FUNCTION_BLOCK FB_StartPos
VAR_INPUT
	bEnable 		: BOOL;
	fCurrentPos 	: LREAL;
END_VAR
VAR_OUTPUT
	fStartPos 		: LREAL;
END_VAR
VAR
END_VAR

IF bEnable THEN
	fStartPos := fStartPos;
	
ELSE 
	fStartPos := fCurrentPos;
END_IF

END_FUNCTION_BLOCK

(* stored: Version 1.1.0.1, ProductVersion 3.1.4024.12
   POU FB_StartPos: Id {203bf98e-10b5-4dfe-b4b1-6b85dd4fc245}, SpecialFunc None *)
